// TwinCAT 3 PLC project FMBasicDevices
// Title: FM Basic Devices
// Company: FrameworkMonorepo
// ProjectVersion: 0.0.1
// ProgramVersion: 3.1.4024.0
// libraries:
//   FM Common Interfaces, * (FrameworkMonorepo)
//   FM Time, * (FrameworkMonorepo)
//   Tc2_Standard, * (Beckhoff Automation GmbH)
// project tree:
//   Beacon/ Beacon.TcPOU, BeaconItem.TcDUT, BeaconParameters.TcGVL
//   Button/ Button.TcPOU
//   Version/ Global_Version.TcGVL
// (motion and I/O tree: see PLC project fmtypes)
// real-time tasks:
//   TASK BindingTestTask: cycle T#1ms, priority 20, ADS port 350
//   TASK PlcTask: cycle T#1ms, priority 21, ADS port 351
//   TASK PlcTask1: cycle T#1ms, priority 22, ADS port 352
//   TASK PlcTask2: cycle T#1ms, priority 23, ADS port 353
//   TASK MathTestTask: cycle T#1ms, priority 24, ADS port 354
//   TASK TimesTestsTask: cycle T#1ms, priority 25, ADS port 355

// ---- Beacon/BeaconItem.TcDUT
TYPE BeaconItem :
STRUCT
	Number : INT;
	Clock : Clock;
	Output : REFERENCE TO BOOL;
	Duration : TON;
	DurationTime : TIME;
END_STRUCT
END_TYPE

// ---- Beacon/BeaconParameters.TcGVL
{attribute 'qualified_only'}
VAR_GLOBAL CONSTANT
	MaxColorCount : INT := 4;
END_VAR

// ---- Version/Global_Version.TcGVL
{attribute 'TcGenerated'}
{attribute 'no-analysis'}
{attribute 'linkalways'}
// This function has been automatically generated from the project information.
VAR_GLOBAL CONSTANT
	{attribute 'const_non_replaced'}
	stLibVersion_FM_Basic_Devices : ST_LibVersion := (iMajor := 0, iMinor := 0, iBuild := 1, iRevision := 0, nFlags := 0, sVersion := '0.0.1');
END_VAR

// ---- Beacon/Beacon.TcPOU
FUNCTION_BLOCK Beacon IMPLEMENTS Cyclic
VAR
	colors : ARRAY[0..MaxColorCount - 1] OF BeaconItem;
	definedColors : INT;
END_VAR
VAR CONSTANT
	MaxColorCount : INT := BeaconParameters.MaxColorCount;
END_VAR

METHOD Blink
VAR_INPUT
	color : INT;
	period : TIME;
END_VAR
VAR
	item : REFERENCE TO BeaconItem;
END_VAR
item REF= GetColor(color);
IF (NOT __ISVALIDREF(item)) THEN
	RETURN;
END_IF

item.Clock.Enable := TRUE;
item.Clock.Period := period;

item.Duration(IN := FALSE);
item.DurationTime := T#0S;
END_METHOD

METHOD Cyclic
VAR
	i : INT;
	color : REFERENCE TO BeaconItem;
END_VAR
FOR i := 0 TO definedColors - 1 DO
	color REF= colors[i];
	color.Clock.Cyclic();
	color.Output := color.Clock.Clock;
	color.Duration();
	IF (color.Duration.Q AND color.DurationTime > T#0S) THEN
		Off(i);
		color.Duration(IN := FALSE);
	END_IF
END_FOR
END_METHOD

METHOD DefineColor
VAR_INPUT
	ColorEnum : INT; // Create enum for this
	Output : REFERENCE TO BOOL;
END_VAR
IF (definedColors < MaxColorCount) THEN
	colors[definedColors].Number := ColorEnum;
	colors[definedColors].Output REF= Output;
	definedColors := definedColors + 1;
END_IF
END_METHOD

METHOD ForTime
VAR_INPUT
	color : INT;
	duration : TIME;
END_VAR
VAR
	item : REFERENCE TO BeaconItem;
END_VAR
item REF= GetColor(color);
IF (NOT __ISVALIDREF(item)) THEN
	RETURN;
END_IF

item.Duration(IN := FALSE);
item.Duration(IN := TRUE, PT := duration);
item.DurationTime := duration;
END_METHOD

METHOD GetColor : REFERENCE TO BeaconItem
VAR_INPUT
	number : INT;
END_VAR
VAR
	i : INT;
END_VAR
FOR i := 0 TO definedColors - 1 DO
	IF (colors[i].Number = number) THEN
		GetColor REF= colors[i];
		RETURN;
	END_IF
END_FOR
END_METHOD

METHOD Light
VAR_INPUT
	color : INT;
END_VAR
VAR
	item : REFERENCE TO BeaconItem;
END_VAR
item REF= GetColor(color);
IF (NOT __ISVALIDREF(item)) THEN
	RETURN;
END_IF

item.Clock.Enable := TRUE;
item.Clock.Period := T#0S;

item.Duration(IN := FALSE);
item.DurationTime := T#0S;
END_METHOD

METHOD Off
VAR_INPUT
	color : INT;
END_VAR
VAR
	item : REFERENCE TO BeaconItem;
END_VAR
item REF= GetColor(color);
IF (NOT __ISVALIDREF(item)) THEN
	RETURN;
END_IF

item.Clock.Enable := FALSE;

item.Duration(IN := FALSE);
item.DurationTime := T#0S;
END_METHOD

METHOD SetBlinkDuty
VAR_INPUT
	color : INT;
	duty : LREAL;
END_VAR
VAR
	item : REFERENCE TO BeaconItem;
END_VAR
item REF= GetColor(color);
IF (NOT __ISVALIDREF(item)) THEN
	RETURN;
END_IF

item.Clock.Duty := duty;
END_METHOD

END_FUNCTION_BLOCK

// ---- Button/Button.TcPOU
FUNCTION_BLOCK Button IMPLEMENTS Cyclic
VAR
	button : REFERENCE TO BOOL;
	
	filter : TON;
	pressTrigger : R_TRIG;
	
	_FilterTime : TIME := T#100MS;
END_VAR

METHOD Cyclic
filter(IN := button, PT := _FilterTime);
pressTrigger(CLK := filter.Q);
END_METHOD

METHOD FB_init : BOOL
VAR_INPUT
	bInitRetains : BOOL; // if TRUE, the retain variables are initialized (warm start / cold start)
	bInCopyCode : BOOL;  // if TRUE, the instance afterwards gets moved into the copy code (online change)
	
	button : REFERENCE TO BOOL;
END_VAR
THIS^.button REF= button;
END_METHOD

{attribute 'monitoring' := 'call'}
PROPERTY FilterTime : TIME
GET
FilterTime := _FilterTime;
END_GET
SET
_FilterTime := FilterTime;
END_SET
END_PROPERTY

{attribute 'monitoring' := 'call'}
PROPERTY JustPressed : BOOL
GET
JustPressed := pressTrigger.Q;
END_GET
END_PROPERTY

{attribute 'monitoring' := 'call'}
PROPERTY Pressed : BOOL
GET
Pressed := filter.Q;
END_GET
END_PROPERTY

END_FUNCTION_BLOCK
